(* LS Electric XG5000 project: 02_04_Practice2 *)
(* PLC LSPLC *)
(* module base 0 slot 0: 입력 모듈:XGI-D21A (DC 24V 입력, 8점 (전류소스/싱크입력)) *)
(* module base 0 slot 1: 출력 모듈:XGQ-RY1A (릴레이 출력, 8점 (2A용, 단독 COM.)) *)

PROGRAM NewProgram (* task: 스캔 프로그램 *)
VAR
    역방향입력 AT %IX0.0.2 : BOOL;
    역방향회전 AT %QX0.1.1 : BOOL;
    정방향입력 AT %IX0.0.1 : BOOL;
    정방향회전 AT %QX0.1.0 : BOOL;
    정지버튼 AT %IX0.0.0 : BOOL;
END_VAR

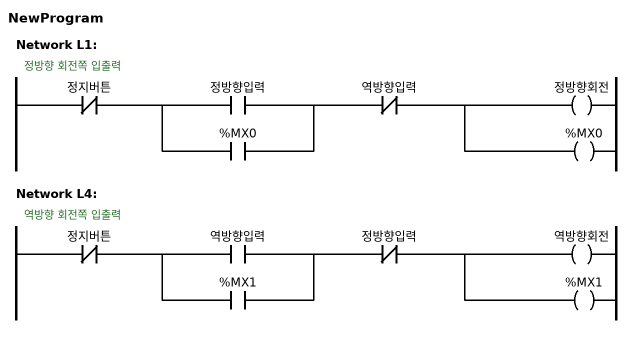
(* 정방향 회전쪽 입출력 *)
(* Rung L1 *)
정방향회전 := NOT 정지버튼 AND (정방향입력 OR %MX0) AND NOT 역방향입력;
%MX0 := NOT 정지버튼 AND (정방향입력 OR %MX0) AND NOT 역방향입력;
(* 역방향 회전쪽 입출력 *)
(* Rung L4 *)
역방향회전 := NOT 정지버튼 AND (역방향입력 OR %MX1) AND NOT 정방향입력;
%MX1 := NOT 정지버튼 AND (역방향입력 OR %MX1) AND NOT 정방향입력;
END_PROGRAM